DATA_BLOCK "检修控制_DB"
{ S7_Optimized_Access := 'TRUE' }
VERSION : 0.1
NON_RETAIN
"检修控制"

BEGIN

END_DATA_BLOCK

